// Mitsubishi GX Works2 project: counter basic   PLC: FX1N/FX1NC

PROGRAM MAIN
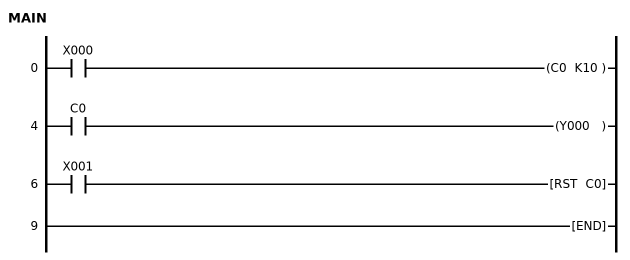
0     LD      X000
      OUT     C0 K10
4     LD      C0
      OUT     Y000
6     LD      X001
      RST     C0
9     END
END_PROGRAM
